Staubli VAL3: initdata.pgx

program initdata()
begin
  nTxtTotal=11
  nNumTotal=5031
  n_sTxt=0
  nNumrecord=0
  fout=true
  bSignal=false
  bTxt1=false
  bTxt2=false
  bTxt3=false
  btrig=true
  call Txt_initData()
  call txt_PkgInit()

  //clearBuffer(sSocketout)
  //sioSet(sSocketout,nByteOut)
end
